(* IEC 61131-3 sources: sigmatek-logger-api/IXON_API/Class/cIXONConv5Int5Str, 1 file *)

(* ---- cIXONConv5Int5Str.st ---- *)
#DEFINE MAX_NAME_LENGTH 100
#DEFINE MAX_INTEGER_LENGTH 10
#DEFINE MAX_DATASTRING_LENGTH 1024
#DEFINE MAX_STRING_LENGTH 100

(*!
<Class
	Name               = "cIXONConv5Int5Str"
	Revision           = "0.0"
	RealtimeTask       = "false"
	CyclicTask         = "false"
	BackgroundTask     = "false"
	Sigmatek           = "false"
	OSInterface        = "false"
	HighPriority       = "false"
	Automatic          = "false"
	UpdateMode         = "Prescan"
	SharedCommandTable = "true"
	Objectsize         = "(510,120)">
	<Channels>
		<Server Name="ClassSvr" Visualized="false" Initialize="false" WriteProtected="true" Retentive="false"/>
		<Server Name="sCmdConvert" Visualized="false" Initialize="false" WriteProtected="false" Retentive="false"/>
		<Server Name="sInteger1" Visualized="false" Initialize="false" WriteProtected="false" Retentive="false"/>
		<Server Name="sInteger2" Visualized="false" Initialize="false" WriteProtected="false" Retentive="false"/>
		<Server Name="sInteger3" Visualized="false" Initialize="false" WriteProtected="false" Retentive="false"/>
		<Server Name="sInteger4" Visualized="false" Initialize="false" WriteProtected="false" Retentive="false"/>
		<Server Name="sInteger5" Visualized="false" Initialize="false" WriteProtected="false" Retentive="false"/>
		<Server Name="sIntegerName1" Class="String" Visualized="true" Initialize="true" WriteProtected="false" Retentive="false"/>
		<Server Name="sIntegerName2" Class="String" Visualized="true" Initialize="true" WriteProtected="false" Retentive="false"/>
		<Server Name="sIntegerName3" Class="String" Visualized="true" Initialize="true" WriteProtected="false" Retentive="false"/>
		<Server Name="sIntegerName4" Class="String" Visualized="true" Initialize="true" WriteProtected="false" Retentive="false"/>
		<Server Name="sIntegerName5" Class="String" Visualized="true" Initialize="true" WriteProtected="false" Retentive="false"/>
		<Server Name="sSetInitNrOfInteger" Visualized="false" Initialize="true" DefValue="1" WriteProtected="true" Retentive="false"/>
		<Server Name="sSetInitNrOfString" Visualized="false" Initialize="true" DefValue="1" WriteProtected="true" Retentive="false"/>
		<Server Name="sString1" Class="String" Visualized="false" Initialize="true" WriteProtected="false" Retentive="false"/>
		<Server Name="sString2" Class="String" Visualized="false" Initialize="true" WriteProtected="false" Retentive="false"/>
		<Server Name="sString3" Class="String" Visualized="false" Initialize="true" WriteProtected="false" Retentive="false"/>
		<Server Name="sString4" Class="String" Visualized="false" Initialize="true" WriteProtected="false" Retentive="false"/>
		<Server Name="sString5" Class="String" Visualized="false" Initialize="true" WriteProtected="false" Retentive="false"/>
		<Server Name="sStringName1" Class="String" Visualized="true" Initialize="true" WriteProtected="false" Retentive="false"/>
		<Server Name="sStringName2" Class="String" Visualized="true" Initialize="true" WriteProtected="false" Retentive="false"/>
		<Server Name="sStringName3" Class="String" Visualized="true" Initialize="true" WriteProtected="false" Retentive="false"/>
		<Server Name="sStringName4" Class="String" Visualized="true" Initialize="true" WriteProtected="false" Retentive="false"/>
		<Server Name="sStringName5" Class="String" Visualized="true" Initialize="true" WriteProtected="false" Retentive="false"/>
		<Server Name="sTriggerName" Class="String" Visualized="false" Initialize="true" WriteProtected="true" Retentive="false"/>
		<Client Name="IntegerName1" Required="true" Internal="true"/>
		<Client Name="IntegerName2" Required="true" Internal="true"/>
		<Client Name="IntegerName3" Required="true" Internal="true"/>
		<Client Name="IntegerName4" Required="true" Internal="true"/>
		<Client Name="IntegerName5" Required="true" Internal="true"/>
		<Client Name="ocSigCLib" Required="false" Internal="false"/>
		<Client Name="String1" Required="true" Internal="true"/>
		<Client Name="String2" Required="true" Internal="true"/>
		<Client Name="String3" Required="true" Internal="true"/>
		<Client Name="String4" Required="true" Internal="true"/>
		<Client Name="String5" Required="true" Internal="true"/>
		<Client Name="StringName1" Required="true" Internal="true"/>
		<Client Name="StringName2" Required="true" Internal="true"/>
		<Client Name="StringName3" Required="true" Internal="true"/>
		<Client Name="StringName4" Required="true" Internal="true"/>
		<Client Name="StringName5" Required="true" Internal="true"/>
		<Client Name="ToIXON_LoggerAPI" Required="true" Internal="false"/>
		<Client Name="TriggerName" Required="true" Internal="true"/>
	</Channels>
	<Separators>
		<Servers>
			<SepChn Position="6"/>
			<SepChn Position="17"/>
			<SepChn Position="4"/>
		</Servers>
	</Separators>
	<Network Name="cIXONConv5Int5Str">
		<!-- List of Components in this network -->
		<Components>
			<Object
				Name       = "IntegerName1"
				Class      = "String"
				Position   = "(750,300)"
				Visualized = "true"
				Remotely   = "true">
				<Channels>
					<Server Name="Data"/>
					<Client Name="SingleRealloc" Value="1"/>
				</Channels>
			</Object>
			<Object
				Name       = "IntegerName2"
				Class      = "String"
				Position   = "(750,450)"
				Visualized = "true"
				Remotely   = "true">
				<Channels>
					<Server Name="Data"/>
					<Client Name="SingleRealloc" Value="1"/>
				</Channels>
			</Object>
			<Object
				Name       = "IntegerName3"
				Class      = "String"
				Position   = "(750,600)"
				Visualized = "true"
				Remotely   = "true">
				<Channels>
					<Server Name="Data"/>
					<Client Name="SingleRealloc" Value="1"/>
				</Channels>
			</Object>
			<Object
				Name       = "IntegerName4"
				Class      = "String"
				Position   = "(750,750)"
				Visualized = "true"
				Remotely   = "true">
				<Channels>
					<Server Name="Data"/>
					<Client Name="SingleRealloc" Value="1"/>
				</Channels>
			</Object>
			<Object
				Name       = "IntegerName5"
				Class      = "String"
				Position   = "(750,900)"
				Visualized = "true"
				Remotely   = "true">
				<Channels>
					<Server Name="Data"/>
					<Client Name="SingleRealloc" Value="1"/>
				</Channels>
			</Object>
			<Object
				Name       = "String1"
				Class      = "String"
				Position   = "(270,1050)"
				Visualized = "true"
				Remotely   = "true">
				<Channels>
					<Server Name="Data"/>
					<Client Name="SingleRealloc" Value="1"/>
				</Channels>
			</Object>
			<Object
				Name       = "String2"
				Class      = "String"
				Position   = "(270,1200)"
				Visualized = "true"
				Remotely   = "true">
				<Channels>
					<Server Name="Data"/>
					<Client Name="SingleRealloc" Value="1"/>
				</Channels>
			</Object>
			<Object
				Name       = "String3"
				Class      = "String"
				Position   = "(270,1350)"
				Visualized = "true"
				Remotely   = "true">
				<Channels>
					<Server Name="Data"/>
					<Client Name="SingleRealloc" Value="1"/>
				</Channels>
			</Object>
			<Object
				Name       = "String4"
				Class      = "String"
				Position   = "(270,1500)"
				Visualized = "true"
				Remotely   = "true">
				<Channels>
					<Server Name="Data"/>
					<Client Name="SingleRealloc" Value="1"/>
				</Channels>
			</Object>
			<Object
				Name       = "String5"
				Class      = "String"
				Position   = "(270,1650)"
				Visualized = "true"
				Remotely   = "true">
				<Channels>
					<Server Name="Data"/>
					<Client Name="SingleRealloc" Value="1"/>
				</Channels>
			</Object>
			<Object
				Name       = "StringName1"
				Class      = "String"
				Position   = "(750,1050)"
				Visualized = "true"
				Remotely   = "true">
				<Channels>
					<Server Name="Data"/>
					<Client Name="SingleRealloc" Value="1"/>
				</Channels>
			</Object>
			<Object
				Name       = "StringName2"
				Class      = "String"
				Position   = "(750,1200)"
				Visualized = "true"
				Remotely   = "true">
				<Channels>
					<Server Name="Data"/>
					<Client Name="SingleRealloc" Value="1"/>
				</Channels>
			</Object>
			<Object
				Name       = "StringName3"
				Class      = "String"
				Position   = "(750,1350)"
				Visualized = "true"
				Remotely   = "true">
				<Channels>
					<Server Name="Data"/>
					<Client Name="SingleRealloc" Value="1"/>
				</Channels>
			</Object>
			<Object
				Name       = "StringName4"
				Class      = "String"
				Position   = "(750,1500)"
				Visualized = "true"
				Remotely   = "true">
				<Channels>
					<Server Name="Data"/>
					<Client Name="SingleRealloc" Value="1"/>
				</Channels>
			</Object>
			<Object
				Name       = "StringName5"
				Class      = "String"
				Position   = "(750,1650)"
				Visualized = "true"
				Remotely   = "true">
				<Channels>
					<Server Name="Data"/>
					<Client Name="SingleRealloc" Value="1"/>
				</Channels>
			</Object>
			<Object
				Name       = "TriggerName"
				Class      = "String"
				Position   = "(750,150)"
				Visualized = "true"
				Remotely   = "true">
				<Channels>
					<Server Name="Data"/>
					<Client Name="SingleRealloc" Value="1"/>
				</Channels>
			</Object>
		</Components>
		<Comments>
		</Comments>
		<!-- List of Connections in this network -->
		<Connections>
			<Connection Source="this.TriggerName" Destination="TriggerName.Data"/>
			<Connection Source="this.sTriggerName" Destination="TriggerName.Data" Vertices="(1298,390),(1126,240),"/>
			<Connection Source="this.IntegerName1" Destination="IntegerName1.Data"/>
			<Connection Source="this.sIntegerName1" Destination="IntegerName1.Data" Vertices="(1298,510),(1126,390),"/>
			<Connection Source="this.IntegerName2" Destination="IntegerName2.Data"/>
			<Connection Source="this.sIntegerName2" Destination="IntegerName2.Data" Vertices="(1298,630),(1126,540),"/>
			<Connection Source="this.IntegerName3" Destination="IntegerName3.Data"/>
			<Connection Source="this.IntegerName4" Destination="IntegerName4.Data"/>
			<Connection Source="this.IntegerName5" Destination="IntegerName5.Data"/>
			<Connection Source="this.sIntegerName3" Destination="IntegerName3.Data" Vertices="(1298,750),(1126,690),"/>
			<Connection Source="this.sIntegerName4" Destination="IntegerName4.Data" Vertices="(1298,870),(1126,840),"/>
			<Connection Source="this.StringName1" Destination="StringName1.Data"/>
			<Connection Source="this.StringName2" Destination="StringName2.Data"/>
			<Connection Source="this.sIntegerName5" Destination="IntegerName5.Data" Vertices="(1298,990),(1126,990),"/>
			<Connection Source="this.sStringName1" Destination="StringName1.Data" Vertices="(1298,1110),(1126,1140),"/>
			<Connection Source="this.sStringName2" Destination="StringName2.Data" Vertices="(1298,1230),(1126,1290),"/>
			<Connection Source="this.StringName3" Destination="StringName3.Data"/>
			<Connection Source="this.StringName4" Destination="StringName4.Data"/>
			<Connection Source="this.StringName5" Destination="StringName5.Data"/>
			<Connection Source="this.sStringName3" Destination="StringName3.Data" Vertices="(1298,1350),(1126,1440),"/>
			<Connection Source="this.sStringName4" Destination="StringName4.Data" Vertices="(1298,1470),(1126,1590),"/>
			<Connection Source="this.sStringName5" Destination="StringName5.Data" Vertices="(1298,1590),(1126,1740),"/>
			<Connection Source="this.String1" Destination="String1.Data"/>
			<Connection Source="this.sString1" Destination="String1.Data" Vertices="(1298,1170),(646,1140),"/>
			<Connection Source="this.String2" Destination="String2.Data"/>
			<Connection Source="this.String3" Destination="String3.Data"/>
			<Connection Source="this.String4" Destination="String4.Data"/>
			<Connection Source="this.String5" Destination="String5.Data"/>
			<Connection Source="this.sString5" Destination="String5.Data" Vertices="(1298,1650),(646,1740),"/>
			<Connection Source="this.sString2" Destination="String2.Data" Vertices="(1298,1290),(646,1290),"/>
			<Connection Source="this.sString3" Destination="String3.Data" Vertices="(1298,1410),(646,1440),"/>
			<Connection Source="this.sString4" Destination="String4.Data" Vertices="(1298,1530),(646,1590),"/>
		</Connections>
		<!-- Headerfiles -->
		<Options>
		</Options>
	</Network>
</Class>
*)
cIXONConv5Int5Str : CLASS
  //Servers:
	ClassSvr 	: SvrChCmd_DINT;
	sSetInitNrOfInteger 	: SvrCh_UDINT;
	sSetInitNrOfString 	: SvrCh_UDINT;
	sTriggerName 	: SvrChCmd_UDINT;
	sCmdConvert 	: SvrCh_DINT;
	sIntegerName1 	: SvrChCmd_UDINT;
	sInteger1 	: SvrCh_DINT;
	sIntegerName2 	: SvrChCmd_UDINT;
	sInteger2 	: SvrCh_DINT;
	sIntegerName3 	: SvrChCmd_UDINT;
	sInteger3 	: SvrCh_DINT;
	sIntegerName4 	: SvrChCmd_UDINT;
	sInteger4 	: SvrCh_DINT;
	sIntegerName5 	: SvrChCmd_UDINT;
	sInteger5 	: SvrCh_DINT;
	sStringName1 	: SvrChCmd_UDINT;
	sString1 	: SvrChCmd_UDINT;
	sStringName2 	: SvrChCmd_UDINT;
	sString2 	: SvrChCmd_UDINT;
	sStringName3 	: SvrChCmd_UDINT;
	sString3 	: SvrChCmd_UDINT;
	sStringName4 	: SvrChCmd_UDINT;
	sString4 	: SvrChCmd_UDINT;
	sStringName5 	: SvrChCmd_UDINT;
	sString5 	: SvrChCmd_UDINT;
  //Clients:
	ToIXON_LoggerAPI 	: CltChCmd_IXON_LoggerAPI_Interface;
	ocSigCLib 	: CltChCmd_SigCLib;
	TriggerName 	: CltChCmd_String;
	String1 	: CltChCmd_String;
	String2 	: CltChCmd_String;
	String3 	: CltChCmd_String;
	String4 	: CltChCmd_String;
	String5 	: CltChCmd_String;
	IntegerName1 	: CltChCmd_String;
	IntegerName2 	: CltChCmd_String;
	IntegerName3 	: CltChCmd_String;
	IntegerName4 	: CltChCmd_String;
	IntegerName5 	: CltChCmd_String;
	StringName1 	: CltChCmd_String;
	StringName2 	: CltChCmd_String;
	StringName3 	: CltChCmd_String;
	StringName4 	: CltChCmd_String;
	StringName5 	: CltChCmd_String;
  //Variables:
		vNameString : ARRAY [0..MAX_NAME_LENGTH-1] OF CHAR;

		vIntValueString : ARRAY [0..MAX_INTEGER_LENGTH-1] OF CHAR;

		vStrValueString : ARRAY [0..MAX_STRING_LENGTH-1] OF CHAR;

		vDataString : ARRAY [0..MAX_DATASTRING_LENGTH-1] OF CHAR;

  //Functions:

	FUNCTION BuildConfigString;

	FUNCTION BuildPairInteger
		VAR_INPUT
			Value 	: DINT;
		END_VAR;

	FUNCTION BuildPairString;

	FUNCTION BuildTrigger
		VAR_INPUT
			Value 	: DINT;
		END_VAR;

	FUNCTION VIRTUAL GLOBAL sTriggerName::Read
		VAR_OUTPUT
			output (EAX) 	: UDINT;
		END_VAR;

	FUNCTION VIRTUAL GLOBAL sTriggerName::Write
		VAR_INPUT
			input (EAX) 	: UDINT;
		END_VAR
		VAR_OUTPUT
			result (EAX) 	: UDINT;
		END_VAR;

	FUNCTION VIRTUAL GLOBAL sCmdConvert::Write
		VAR_INPUT
			input (EAX) 	: DINT;
		END_VAR
		VAR_OUTPUT
			result (EAX) 	: DINT;
		END_VAR;

	FUNCTION VIRTUAL GLOBAL sIntegerName1::Read
		VAR_OUTPUT
			output (EAX) 	: UDINT;
		END_VAR;

	FUNCTION VIRTUAL GLOBAL sIntegerName1::Write
		VAR_INPUT
			input (EAX) 	: UDINT;
		END_VAR
		VAR_OUTPUT
			result (EAX) 	: UDINT;
		END_VAR;

	FUNCTION VIRTUAL GLOBAL sIntegerName2::Read
		VAR_OUTPUT
			output (EAX) 	: UDINT;
		END_VAR;

	FUNCTION VIRTUAL GLOBAL sIntegerName2::Write
		VAR_INPUT
			input (EAX) 	: UDINT;
		END_VAR
		VAR_OUTPUT
			result (EAX) 	: UDINT;
		END_VAR;

	FUNCTION VIRTUAL GLOBAL sIntegerName3::Read
		VAR_OUTPUT
			output (EAX) 	: UDINT;
		END_VAR;

	FUNCTION VIRTUAL GLOBAL sIntegerName3::Write
		VAR_INPUT
			input (EAX) 	: UDINT;
		END_VAR
		VAR_OUTPUT
			result (EAX) 	: UDINT;
		END_VAR;

	FUNCTION VIRTUAL GLOBAL sIntegerName4::Read
		VAR_OUTPUT
			output (EAX) 	: UDINT;
		END_VAR;

	FUNCTION VIRTUAL GLOBAL sIntegerName4::Write
		VAR_INPUT
			input (EAX) 	: UDINT;
		END_VAR
		VAR_OUTPUT
			result (EAX) 	: UDINT;
		END_VAR;

	FUNCTION VIRTUAL GLOBAL sIntegerName5::Read
		VAR_OUTPUT
			output (EAX) 	: UDINT;
		END_VAR;

	FUNCTION VIRTUAL GLOBAL sIntegerName5::Write
		VAR_INPUT
			input (EAX) 	: UDINT;
		END_VAR
		VAR_OUTPUT
			result (EAX) 	: UDINT;
		END_VAR;

	FUNCTION VIRTUAL GLOBAL sStringName1::Read
		VAR_OUTPUT
			output (EAX) 	: UDINT;
		END_VAR;

	FUNCTION VIRTUAL GLOBAL sStringName1::Write
		VAR_INPUT
			input (EAX) 	: UDINT;
		END_VAR
		VAR_OUTPUT
			result (EAX) 	: UDINT;
		END_VAR;

	FUNCTION VIRTUAL GLOBAL sString1::Read
		VAR_OUTPUT
			output (EAX) 	: UDINT;
		END_VAR;

	FUNCTION VIRTUAL GLOBAL sString1::Write
		VAR_INPUT
			input (EAX) 	: UDINT;
		END_VAR
		VAR_OUTPUT
			result (EAX) 	: UDINT;
		END_VAR;

	FUNCTION VIRTUAL GLOBAL sStringName2::Read
		VAR_OUTPUT
			output (EAX) 	: UDINT;
		END_VAR;

	FUNCTION VIRTUAL GLOBAL sStringName2::Write
		VAR_INPUT
			input (EAX) 	: UDINT;
		END_VAR
		VAR_OUTPUT
			result (EAX) 	: UDINT;
		END_VAR;

	FUNCTION VIRTUAL GLOBAL sString2::Read
		VAR_OUTPUT
			output (EAX) 	: UDINT;
		END_VAR;

	FUNCTION VIRTUAL GLOBAL sString2::Write
		VAR_INPUT
			input (EAX) 	: UDINT;
		END_VAR
		VAR_OUTPUT
			result (EAX) 	: UDINT;
		END_VAR;

	FUNCTION VIRTUAL GLOBAL sStringName3::Read
		VAR_OUTPUT
			output (EAX) 	: UDINT;
		END_VAR;

	FUNCTION VIRTUAL GLOBAL sStringName3::Write
		VAR_INPUT
			input (EAX) 	: UDINT;
		END_VAR
		VAR_OUTPUT
			result (EAX) 	: UDINT;
		END_VAR;

	FUNCTION VIRTUAL GLOBAL sString3::Read
		VAR_OUTPUT
			output (EAX) 	: UDINT;
		END_VAR;

	FUNCTION VIRTUAL GLOBAL sString3::Write
		VAR_INPUT
			input (EAX) 	: UDINT;
		END_VAR
		VAR_OUTPUT
			result (EAX) 	: UDINT;
		END_VAR;

	FUNCTION VIRTUAL GLOBAL sStringName4::Read
		VAR_OUTPUT
			output (EAX) 	: UDINT;
		END_VAR;

	FUNCTION VIRTUAL GLOBAL sStringName4::Write
		VAR_INPUT
			input (EAX) 	: UDINT;
		END_VAR
		VAR_OUTPUT
			result (EAX) 	: UDINT;
		END_VAR;

	FUNCTION VIRTUAL GLOBAL sString4::Read
		VAR_OUTPUT
			output (EAX) 	: UDINT;
		END_VAR;

	FUNCTION VIRTUAL GLOBAL sString4::Write
		VAR_INPUT
			input (EAX) 	: UDINT;
		END_VAR
		VAR_OUTPUT
			result (EAX) 	: UDINT;
		END_VAR;

	FUNCTION VIRTUAL GLOBAL sStringName5::Read
		VAR_OUTPUT
			output (EAX) 	: UDINT;
		END_VAR;

	FUNCTION VIRTUAL GLOBAL sStringName5::Write
		VAR_INPUT
			input (EAX) 	: UDINT;
		END_VAR
		VAR_OUTPUT
			result (EAX) 	: UDINT;
		END_VAR;

	FUNCTION VIRTUAL GLOBAL sString5::Read
		VAR_OUTPUT
			output (EAX) 	: UDINT;
		END_VAR;

	FUNCTION VIRTUAL GLOBAL sString5::Write
		VAR_INPUT
			input (EAX) 	: UDINT;
		END_VAR
		VAR_OUTPUT
			result (EAX) 	: UDINT;
		END_VAR;
  //Tables:
	FUNCTION @STD
		VAR_OUTPUT
			ret_code	: CONFSTATES;
		END_VAR;
	FUNCTION GLOBAL TAB @CT_;
END_CLASS;

#pragma using String
#pragma usingLtd IXON_LoggerAPI_Interface
#pragma usingLtd SigCLib

FUNCTION cIXONConv5Int5Str::BuildConfigString
  VAR
    i : int;
    lValue : dint;
    length : udint;
  END_VAR

  if  sSetInitNrOfInteger > 5
  then
      sSetInitNrOfInteger := 5;
  end_if;

  if  sSetInitNrOfString > 5
  then
      sSetInitNrOfString := 5;
  end_if;

  _memset(dest:=#vDataString, usByte:=16#00, cntr:=MAX_DATASTRING_LENGTH);

  //Write trigger to 1 / true
  TriggerName.TxtGet(pdst :=  #vNameString[0], dstsize := sizeof(vNameString) - 1);
  BuildTrigger(Value := 1);

  //Setup JSON Object Pairs
  for i := 1  to to_int(sSetInitNrOfInteger) do
    //Get Name
    case i of
      1: IntegerName1.TxtGet(pdst := #vNameString[0], dstsize := sizeof(vNameString) - 1);
         lvalue := sInteger1;
      2: IntegerName2.TxtGet(pdst := #vNameString[0], dstsize := sizeof(vNameString) - 1);
         lvalue := sInteger2;
      3: IntegerName3.TxtGet(pdst := #vNameString[0], dstsize := sizeof(vNameString) - 1);
         lvalue := sInteger3;
      4: IntegerName4.TxtGet(pdst := #vNameString[0], dstsize := sizeof(vNameString) - 1);
         lvalue := sInteger4;
      5: IntegerName5.TxtGet(pdst := #vNameString[0], dstsize := sizeof(vNameString) - 1);
         lvalue := sInteger5;
    end_case;

    BuildPairInteger(Value := lValue);

  end_for;

  for i := 1  to to_int(sSetInitNrOfString) do
    case i of
      1: StringName1.TxtGet(pdst := #vNameString[0], dstsize := sizeof(vNameString) - 1);
         String1.TxtGet(pdst := #vStrValueString[0], dstsize := sizeof(vStrValueString) - 1);
      2: StringName2.TxtGet(pdst := #vNameString[0], dstsize := sizeof(vNameString) - 1);
         String2.TxtGet(pdst := #vStrValueString[0], dstsize := sizeof(vStrValueString) - 1);
      3: StringName3.TxtGet(pdst := #vNameString[0], dstsize := sizeof(vNameString) - 1);
         String3.TxtGet(pdst := #vStrValueString[0], dstsize := sizeof(vStrValueString) - 1);
      4: StringName4.TxtGet(pdst := #vNameString[0], dstsize := sizeof(vNameString) - 1);
         String4.TxtGet(pdst := #vStrValueString[0], dstsize := sizeof(vStrValueString) - 1);
      5: StringName5.TxtGet(pdst := #vNameString[0], dstsize := sizeof(vNameString) - 1);
         String5.TxtGet(pdst := #vStrValueString[0], dstsize := sizeof(vStrValueString) - 1);
    end_case;

    BuildPairString();

  end_for;

  //Write trigger to 0 / false
  TriggerName.TxtGet(pdst :=  #vNameString[0], dstsize := sizeof(vNameString) - 1);
  BuildTrigger(Value := 0);

  length := _strlen(src:=#vDataString[0]);
  ToIXON_LoggerAPI.AddStringToBuffer(pData:=#vDataString[0], udLen:=length + 1);

END_FUNCTION

FUNCTION cIXONConv5Int5Str::BuildPairInteger
	VAR_INPUT
		Value 	: DINT;
	END_VAR
  VAR
  	length : UDINT;
  END_VAR

  ocSigCLib.IToA(val  := to_dint(Value),
                 dst  := #vIntValueString[0],
                 base := 10);

  length := _strlen(src:=#vDataString[0]);
  vDataString[length] := '@';
  _strcat(dest:=#vDataString[length + 1], src:=#vNameString[0]);
  length := _strlen(src:=#vDataString[0]);
  vDataString[length] := '=';
  _strcat(dest:=#vDataString[length + 1], src:=#vIntValueString[0]);
  length := _strlen(src:=#vDataString[0]);
  vDataString[length] := 16#0A;

END_FUNCTION

FUNCTION cIXONConv5Int5Str::BuildPairString
  VAR
  	length : UDINT;
    strLength : UDINT;
  END_VAR

  strLength := _strlen(src:=#vStrValueString[0]);

  length := _strlen(src:=#vDataString[0]);
  vDataString[length] := '@';
  _strcat(dest:=#vDataString[length + 1], src:=#vNameString[0]);
  length := _strlen(src:=#vDataString[0]);
  vDataString[length] := '=';
  ocSigCLib.IToA(val  := to_dint(strLength),
                 dst  := #vDataString[length+1],
                 base := 10);
  length := _strlen(src:=#vDataString[0]);
  vDataString[length] := ',';
  _strcat(dest:=#vDataString[length + 1], src:=#vStrValueString[0]);
  length := _strlen(src:=#vDataString[0]);
  vDataString[length] := 16#0A;

END_FUNCTION

FUNCTION cIXONConv5Int5Str::BuildTrigger
	VAR_INPUT
		Value 	: DINT;
	END_VAR
  VAR
  	length : UDINT;
  END_VAR

  ocSigCLib.IToA(val  := to_dint(Value),
                 dst  := #vIntValueString[0],
                 base := 10);

  length := _strlen(src:=#vDataString[0]);
  vDataString[length] := '@';
  _strcat(dest:=#vDataString[length + 1], src:=#vNameString[0]);
  length := _strlen(src:=#vDataString[0]);
  vDataString[length] := '=';
  if value = 0 then
    vDataString[length + 1] := 'f';
  else
    vDataString[length + 1] := 't';
  end_if;
  vDataString[length + 2] := 16#0A;

END_FUNCTION

FUNCTION VIRTUAL GLOBAL cIXONConv5Int5Str::sCmdConvert::Write
	VAR_INPUT
		input (EAX) 	: DINT;
	END_VAR
	VAR_OUTPUT
		result (EAX) 	: DINT;
	END_VAR

	sCmdConvert := input;
	result := sCmdConvert;

  BuildConfigString();

END_FUNCTION

FUNCTION VIRTUAL GLOBAL cIXONConv5Int5Str::sIntegerName1::Read
	VAR_OUTPUT
		output (EAX) 	: UDINT;
	END_VAR

	sIntegerName1 := IntegerName1.Data.Read();
	output := sIntegerName1;

END_FUNCTION

FUNCTION VIRTUAL GLOBAL cIXONConv5Int5Str::sIntegerName1::Write
	VAR_INPUT
		input (EAX) 	: UDINT;
	END_VAR
	VAR_OUTPUT
		result (EAX) 	: UDINT;
	END_VAR

	sIntegerName1 := input;
	result := (IntegerName1.Data.Write(sIntegerName1))$UDINT;

END_FUNCTION

FUNCTION VIRTUAL GLOBAL cIXONConv5Int5Str::sIntegerName2::Read
	VAR_OUTPUT
		output (EAX) 	: UDINT;
	END_VAR

	sIntegerName2 := IntegerName2.Data.Read();
	output := sIntegerName2;

END_FUNCTION

FUNCTION VIRTUAL GLOBAL cIXONConv5Int5Str::sIntegerName2::Write
	VAR_INPUT
		input (EAX) 	: UDINT;
	END_VAR
	VAR_OUTPUT
		result (EAX) 	: UDINT;
	END_VAR

	sIntegerName2 := input;
	result := (IntegerName2.Data.Write(sIntegerName2))$UDINT;

END_FUNCTION

FUNCTION VIRTUAL GLOBAL cIXONConv5Int5Str::sIntegerName3::Read
	VAR_OUTPUT
		output (EAX) 	: UDINT;
	END_VAR

	sIntegerName3 := IntegerName3.Data.Read();
	output := sIntegerName3;

END_FUNCTION

FUNCTION VIRTUAL GLOBAL cIXONConv5Int5Str::sIntegerName3::Write
	VAR_INPUT
		input (EAX) 	: UDINT;
	END_VAR
	VAR_OUTPUT
		result (EAX) 	: UDINT;
	END_VAR

	sIntegerName3 := input;
	result := (IntegerName3.Data.Write(sIntegerName3))$UDINT;

END_FUNCTION

FUNCTION VIRTUAL GLOBAL cIXONConv5Int5Str::sIntegerName4::Read
	VAR_OUTPUT
		output (EAX) 	: UDINT;
	END_VAR

	sIntegerName4 := IntegerName4.Data.Read();
	output := sIntegerName4;

END_FUNCTION

FUNCTION VIRTUAL GLOBAL cIXONConv5Int5Str::sIntegerName4::Write
	VAR_INPUT
		input (EAX) 	: UDINT;
	END_VAR
	VAR_OUTPUT
		result (EAX) 	: UDINT;
	END_VAR

	sIntegerName4 := input;
	result := (IntegerName4.Data.Write(sIntegerName4))$UDINT;

END_FUNCTION

FUNCTION VIRTUAL GLOBAL cIXONConv5Int5Str::sIntegerName5::Read
	VAR_OUTPUT
		output (EAX) 	: UDINT;
	END_VAR

	sIntegerName5 := IntegerName5.Data.Read();
	output := sIntegerName5;

END_FUNCTION

FUNCTION VIRTUAL GLOBAL cIXONConv5Int5Str::sIntegerName5::Write
	VAR_INPUT
		input (EAX) 	: UDINT;
	END_VAR
	VAR_OUTPUT
		result (EAX) 	: UDINT;
	END_VAR

	sIntegerName5 := input;
	result := (IntegerName5.Data.Write(sIntegerName5))$UDINT;

END_FUNCTION

FUNCTION VIRTUAL GLOBAL cIXONConv5Int5Str::sStringName1::Read
	VAR_OUTPUT
		output (EAX) 	: UDINT;
	END_VAR

	sStringName1 := StringName1.Data.Read();
	output := sStringName1;

END_FUNCTION

FUNCTION VIRTUAL GLOBAL cIXONConv5Int5Str::sStringName1::Write
	VAR_INPUT
		input (EAX) 	: UDINT;
	END_VAR
	VAR_OUTPUT
		result (EAX) 	: UDINT;
	END_VAR

	sStringName1 := input;
	result := (StringName1.Data.Write(sStringName1))$UDINT;

END_FUNCTION

FUNCTION VIRTUAL GLOBAL cIXONConv5Int5Str::sStringName2::Read
	VAR_OUTPUT
		output (EAX) 	: UDINT;
	END_VAR

	sStringName2 := StringName2.Data.Read();
	output := sStringName2;

END_FUNCTION

FUNCTION VIRTUAL GLOBAL cIXONConv5Int5Str::sStringName2::Write
	VAR_INPUT
		input (EAX) 	: UDINT;
	END_VAR
	VAR_OUTPUT
		result (EAX) 	: UDINT;
	END_VAR

	sStringName2 := input;
	result := (StringName2.Data.Write(sStringName2))$UDINT;

END_FUNCTION

FUNCTION VIRTUAL GLOBAL cIXONConv5Int5Str::sStringName3::Read
	VAR_OUTPUT
		output (EAX) 	: UDINT;
	END_VAR

	sStringName3 := StringName3.Data.Read();
	output := sStringName3;

END_FUNCTION

FUNCTION VIRTUAL GLOBAL cIXONConv5Int5Str::sStringName3::Write
	VAR_INPUT
		input (EAX) 	: UDINT;
	END_VAR
	VAR_OUTPUT
		result (EAX) 	: UDINT;
	END_VAR

	sStringName3 := input;
	result := (StringName3.Data.Write(sStringName3))$UDINT;

END_FUNCTION

FUNCTION VIRTUAL GLOBAL cIXONConv5Int5Str::sStringName4::Read
	VAR_OUTPUT
		output (EAX) 	: UDINT;
	END_VAR

	sStringName4 := StringName4.Data.Read();
	output := sStringName4;

END_FUNCTION

FUNCTION VIRTUAL GLOBAL cIXONConv5Int5Str::sStringName4::Write
	VAR_INPUT
		input (EAX) 	: UDINT;
	END_VAR
	VAR_OUTPUT
		result (EAX) 	: UDINT;
	END_VAR

	sStringName4 := input;
	result := (StringName4.Data.Write(sStringName4))$UDINT;

END_FUNCTION

FUNCTION VIRTUAL GLOBAL cIXONConv5Int5Str::sStringName5::Read
	VAR_OUTPUT
		output (EAX) 	: UDINT;
	END_VAR

	sStringName5 := StringName5.Data.Read();
	output := sStringName5;

END_FUNCTION

FUNCTION VIRTUAL GLOBAL cIXONConv5Int5Str::sStringName5::Write
	VAR_INPUT
		input (EAX) 	: UDINT;
	END_VAR
	VAR_OUTPUT
		result (EAX) 	: UDINT;
	END_VAR

	sStringName5 := input;
	result := (StringName5.Data.Write(sStringName5))$UDINT;

END_FUNCTION

FUNCTION VIRTUAL GLOBAL cIXONConv5Int5Str::sTriggerName::Read
	VAR_OUTPUT
		output (EAX) 	: UDINT;
	END_VAR

	sTriggerName := TriggerName.Data.Read();
	output := sTriggerName;

END_FUNCTION

FUNCTION VIRTUAL GLOBAL cIXONConv5Int5Str::sTriggerName::Write
	VAR_INPUT
		input (EAX) 	: UDINT;
	END_VAR
	VAR_OUTPUT
		result (EAX) 	: UDINT;
	END_VAR

	sTriggerName := input;
	result := (TriggerName.Data.Write(sTriggerName))$UDINT;

END_FUNCTION

FUNCTION VIRTUAL GLOBAL cIXONConv5Int5Str::sString1::Read
	VAR_OUTPUT
		output (EAX) 	: UDINT;
	END_VAR

	sString1 := String1.Data.Read();
	output := sString1;

END_FUNCTION

FUNCTION VIRTUAL GLOBAL cIXONConv5Int5Str::sString1::Write
	VAR_INPUT
		input (EAX) 	: UDINT;
	END_VAR
	VAR_OUTPUT
		result (EAX) 	: UDINT;
	END_VAR

	sString1 := input;
	result := (String1.Data.Write(sString1))$UDINT;

END_FUNCTION

FUNCTION VIRTUAL GLOBAL cIXONConv5Int5Str::sString2::Read
	VAR_OUTPUT
		output (EAX) 	: UDINT;
	END_VAR

	sString2 := String2.Data.Read();
	output := sString2;

END_FUNCTION

FUNCTION VIRTUAL GLOBAL cIXONConv5Int5Str::sString2::Write
	VAR_INPUT
		input (EAX) 	: UDINT;
	END_VAR
	VAR_OUTPUT
		result (EAX) 	: UDINT;
	END_VAR

	sString2 := input;
	result := (String2.Data.Write(sString2))$UDINT;

END_FUNCTION

FUNCTION VIRTUAL GLOBAL cIXONConv5Int5Str::sString3::Read
	VAR_OUTPUT
		output (EAX) 	: UDINT;
	END_VAR

	sString3 := String3.Data.Read();
	output := sString3;

END_FUNCTION

FUNCTION VIRTUAL GLOBAL cIXONConv5Int5Str::sString3::Write
	VAR_INPUT
		input (EAX) 	: UDINT;
	END_VAR
	VAR_OUTPUT
		result (EAX) 	: UDINT;
	END_VAR

	sString3 := input;
	result := (String3.Data.Write(sString3))$UDINT;

END_FUNCTION

FUNCTION VIRTUAL GLOBAL cIXONConv5Int5Str::sString4::Read
	VAR_OUTPUT
		output (EAX) 	: UDINT;
	END_VAR

	sString4 := String4.Data.Read();
	output := sString4;

END_FUNCTION

FUNCTION VIRTUAL GLOBAL cIXONConv5Int5Str::sString4::Write
	VAR_INPUT
		input (EAX) 	: UDINT;
	END_VAR
	VAR_OUTPUT
		result (EAX) 	: UDINT;
	END_VAR

	sString4 := input;
	result := (String4.Data.Write(sString4))$UDINT;

END_FUNCTION

FUNCTION VIRTUAL GLOBAL cIXONConv5Int5Str::sString5::Read
	VAR_OUTPUT
		output (EAX) 	: UDINT;
	END_VAR

	sString5 := String5.Data.Read();
	output := sString5;

END_FUNCTION

FUNCTION VIRTUAL GLOBAL cIXONConv5Int5Str::sString5::Write
	VAR_INPUT
		input (EAX) 	: UDINT;
	END_VAR
	VAR_OUTPUT
		result (EAX) 	: UDINT;
	END_VAR

	sString5 := input;
	result := (String5.Data.Write(sString5))$UDINT;

END_FUNCTION
